TYPE T_OnlineChangeTestStage :
STRUCT
	sName: STRING(80);
	nId: UINT;
	iConfiguredFastThread: Stage.I_Thread;
	bFastThreadConfigured: BOOL;
END_STRUCT
END_TYPE

(* stored: Version 1.1.0.1
   DUT T_OnlineChangeTestStage: Id {482f4d8e-7f78-43eb-b0fc-27511399e8ef} *)
